FUNCTION_BLOCK FB_TEST_CheckPartBarcodeFail EXTENDS FB_Test
VAR
END_VAR

METHOD Execute : ST_TestResults
VAR
	MockStatus		: ST_PartStatus;
	fbCell			: FB_Cell;
	testExpected	: BOOL;
	testResult		: BOOL;
END_VAR
MockStatus.bBarcodeStatus := FALSE;
MockStatus.bCapperStatus := TRUE;
MockStatus.bFillerStatus := TRUE;
MockStatus.bWeightStatus := TRUE;

testExpected := FALSE;
testResult := fbCell.CheckPart(MockStatus);

Execute := AssertEquals(
	testExpected, 
	testResult, 
	'Part status fail.'
);
END_METHOD

END_FUNCTION_BLOCK

(* stored: Version 1.1.0.1, ProductVersion 3.1.4024.12
   POU FB_TEST_CheckPartBarcodeFail: Id {8b3115ad-292c-4bb6-86be-84e7df04e518}, SpecialFunc None
   Method Execute: Id {2f575b9c-bd0e-4ea2-922e-4f5ad0595180} *)
